FUNCTION_BLOCK PAEControlModuleBase EXTENDS PAModule IMPLEMENTS IPAControlModule
VAR_INPUT
END_VAR
VAR_OUTPUT
END_VAR
VAR	
	_FaultState : PANotifyState;
	_OperatingTime : TIME;
	_SwitchingFrequency : DINT;
	_TotalAlarms : DINT;
	_TurnOnInstant : DATE_AND_TIME;
	_TurnOffInstant : DATE_AND_TIME;
	_OnTime : TIME;
	_TurnOnDelay : TIME;
	_TurnOffDelay : TIME;
	_FaultDelayTime : TIME;
	_TurnOnInterlockDelay : TIME;
	_DepletingTime : TIME;
	_OnSiteTurnedOn : BOOL;
	_TurnOnInterlock : BOOL;
	_RunningTime : TIME;	
	_IsTriggered : BOOL;
	_FaultStateACK : BOOL;	
	_AllocatedByWay : BYTE;	
	
	// Gibt an, dass dieses Steuerungsmodul gerade von einer Funktion verwendet wird
	_AllocatedByFunction : IPAProcessFunction;
	_RoutingStateThis : PARoutingState;
	_TimerTurnOnDelay : TON;
	_TimerTurnOffDelay : TON;
END_VAR

METHOD PUBLIC AcknowledgeAlarms
VAR_INPUT
END_VAR
END_METHOD

{attribute 'TcRpcEnable'}
PROPERTY PUBLIC AllocatedByFunction : IPAProcessFunction
GET
AllocatedByFunction := _AllocatedByFunction;
END_GET
SET // PUBLIC
_AllocatedByFunction := AllocatedByFunction;
_AllocatedByWay := BOOL_TO_BYTE(_AllocatedByFunction <> 0);
Root.OnPropertyChangedByte(THIS^, 24, _AllocatedByWay);
END_SET
END_PROPERTY

{attribute 'TcRpcEnable'}
PROPERTY PUBLIC AllocatedByWay : BOOL
GET
AllocatedByWay := _AllocatedByFunction <> 0;
END_GET
END_PROPERTY

METHOD PUBLIC CombineRoutingStates : PARoutingState
VAR_INPUT
	direction : PARoutingDirection;
	rStateOfDependents : PARoutingState;
END_VAR
VAR
	rStateCombined : PARoutingState;
END_VAR
IF direction = PARoutingDirection.ToPredecessors THEN
	// TODO: Logik nochmals checken:
	IF rStateOfDependents <= PARoutingState.WaitOnPredecessors THEN
		rStateCombined := PARoutingState.WaitOnPredecessors;
	ELSE
		IF _RoutingStateThis < PARoutingState.PredecessorsFinished THEN
			rStateCombined := PARoutingState.PredecessorsFinished;
		ELSE
			rStateCombined := _RoutingStateThis;
		END_IF
	END_IF
ELSE // direction = PARoutingDirection.ToSuccessors
	IF rStateOfDependents <= PARoutingState.ReachedOnPosition THEN
		rStateCombined := PARoutingState.WaitOnSuccessor;
	ELSE //IF rStateAll >= PARoutingState.RoutePlaced THEN
		IF _RoutingStateThis = PARoutingState.ReachedOnPosition THEN
			rStateCombined := PARoutingState.RoutePlaced;
		ELSIF _RoutingStateThis <= PARoutingState.SuccessorsPlaced THEN
			rStateCombined := PARoutingState.SuccessorsPlaced;
		ELSE
			rStateCombined := _RoutingStateThis;
		END_IF
	END_IF
END_IF

CombineRoutingStates := rStateCombined;
END_METHOD

{attribute 'monitoring' := 'call'}
//{attribute 'TcRpcEnable'}
PROPERTY PUBLIC DepletingTime : TIME
GET
DepletingTime := _DepletingTime;
END_GET
SET
_DepletingTime := DepletingTime;
Root.OnPropertyChangedTime(THIS^, 22, _DepletingTime);
END_SET
END_PROPERTY

{attribute 'monitoring' := 'call'}
//{attribute 'TcRpcEnable'}
PROPERTY PUBLIC FaultDelayTime : TIME
GET
FaultDelayTime := _FaultDelayTime;
END_GET
SET
_FaultDelayTime := FaultDelayTime;
Root.OnPropertyChangedTime(THIS^, 20, _FaultDelayTime);
END_SET
END_PROPERTY

{attribute 'monitoring' := 'call'}
//{attribute 'TcRpcEnable'}
PROPERTY PUBLIC FaultState : PANotifyState
GET
FaultState := _FaultState;
END_GET
SET
_FaultState := FaultState;
Root.OnPropertyChangedInt(THIS^, 23, _FaultState);
END_SET
END_PROPERTY

{attribute 'monitoring' := 'call'}
//{attribute 'TcRpcEnable'}
PROPERTY PUBLIC FaultStateACK : BOOL
GET
FaultStateACK := _FaultStateACK;
END_GET
SET
_FaultStateACK := FaultStateACK;
Root.OnPropertyChangedBool(THIS^, 29, _FaultStateACK);
END_SET
END_PROPERTY

METHOD PUBLIC FB_postinit
VAR_INPUT
		root : IACVariobatch;
END_VAR
SUPER^.FB_postinit(root);
root.OnPropertyChangedTime(THIS^, 12, _OperatingTime);
root.OnPropertyChangedDInt(THIS^, 13, _SwitchingFrequency);
root.OnPropertyChangedDInt(THIS^, 14, _TotalAlarms);
root.OnPropertyChangedDT(THIS^, 15, _TurnOnInstant);
root.OnPropertyChangedDT(THIS^, 16, _TurnOffInstant);
root.OnPropertyChangedTime(THIS^, 17, _OnTime);
root.OnPropertyChangedTime(THIS^, 18, _TurnOnDelay);
root.OnPropertyChangedTime(THIS^, 19, _TurnOffDelay);
root.OnPropertyChangedTime(THIS^, 20, _FaultDelayTime);
root.OnPropertyChangedTime(THIS^, 21, _TurnOnInterlockDelay);
root.OnPropertyChangedTime(THIS^, 22, _DepletingTime);
root.OnPropertyChangedInt(THIS^, 23, _FaultState);
root.OnPropertyChangedByte(THIS^, 24, _AllocatedByWay);
root.OnPropertyChangedBool(THIS^, 25, _OnSiteTurnedOn);
root.OnPropertyChangedBool(THIS^, 26, _TurnOnInterlock);
root.OnPropertyChangedTime(THIS^, 27, _RunningTime);
root.OnPropertyChangedBool(THIS^, 28, _IsTriggered);
root.OnPropertyChangedBool(THIS^, 29, _FaultStateACK);
END_METHOD

// Gibt die Punkte zurück, über die die aktuelle Route gestellt ist bzw. gestellt werden soll
METHOD PUBLIC GetActivePoints : BOOL
VAR_IN_OUT
	resultPoints : ARRAY [1..GCL.cPointMAX] OF IACPoint;
END_VAR
VAR_INPUT
	pointType : PAFindPointType;
END_VAR
VAR
	i: INT;
	j: INT;
	edge : IACEdge;
	rStateAll : PARoutingState;
	iControlModule : IPAControlModule;
END_VAR
IF NOT AllocatedByWay THEN
	GetActivePoints := FALSE;
	RETURN;
END_IF

// Array leeren
FOR i:=1 TO GCL.cPointMAX BY 1
  DO
	resultPoints[i] := 0;
END_FOR;

j := 1;
// Durchlaufe alle Punkte und ermittle den Gesamtstatus über aller Nachfolgeelemente
FOR i:=1 TO GCL.cPointMAX BY 1
  DO
    IF _Points[i] <> 0 THEN
		
	    // Suche aktiven Weg
		edge := _Points[i].GetAllocatedEdge(AllocatedByFunction);
		
		IF edge <> 0 THEN
			IF (pointType = PAFindPointType.InPoints) AND (edge.Target = _Points[i]) THEN
				resultPoints[j] := _Points[i];
			ELSIF (pointType = PAFindPointType.OutPoints) AND (edge.Source = _Points[i]) THEN
				resultPoints[j] := _Points[i];
			ELSE
				resultPoints[j] := _Points[i];			
			END_IF
			j := j + 1;
		END_IF
	ELSE
		EXIT;
	END_IF
END_FOR;

GetActivePoints := TRUE;
RETURN;
END_METHOD

METHOD PUBLIC GetRoutingStateOfDependents : PARoutingState
VAR_IN_OUT
	activeOutPoints : ARRAY [1..GCL.cPointMAX] OF IACPoint;
	activeInPoints : ARRAY [1..GCL.cPointMAX] OF IACPoint;
END_VAR
VAR_INPUT
	direction : PARoutingDirection;
END_VAR
VAR
	i: INT;
	edge : IACEdge;
	rStateAll : PARoutingState;
	iControlModule : IPAControlModule;
	iProcessModule : IPAProcessModule;
	targetRoutingState : PARoutingState;
	findPointType : PAFindPointType;
END_VAR
IF NOT AllocatedByWay THEN
	GetRoutingStateOfDependents := PARoutingState.Idle;
	RETURN;
END_IF

IF direction = PARoutingDirection.ToPredecessors THEN
	findPointType := PAFindPointType.InPoints;
	rStateAll := PARoutingState.ReachedOffPosition;
ELSE // direction = PARoutingDirection.ToSuccessors
	findPointType := PAFindPointType.OutPoints;
	rStateAll := PARoutingState.RoutePlaced;
END_IF

GetActivePoints(activeOutPoints,PAFindPointType.OutPoints);
GetActivePoints(activeInPoints,PAFindPointType.InPoints);

// Durchlaufe alle Punkte und ermittle den Gesamtstatus über alle Elemente
// Falls Suchrichtung zu Nachfolger (Ausgangspunkte)
IF (direction = PARoutingDirection.ToSuccessors) THEN		
	FOR i:=1 TO GCL.cPointMAX BY 1
	  DO
		IF activeOutPoints[i] <> 0 THEN
			
			// Suche aktiven Weg
			edge := activeOutPoints[i].GetAllocatedEdge(AllocatedByFunction);
			
			// Falls das Ziel ein Control-Module ist dann frage Status ab und korrigiere Gesamtstatus aller Nachfolger
			IF __QUERYINTERFACE(edge.Target, iControlModule) THEN
				targetRoutingState := iControlModule.RoutingStateToTarget;
				IF targetRoutingState < rStateAll THEN
					rStateAll := targetRoutingState;
				END_IF
			ELSIF __QUERYINTERFACE(edge.Target, iProcessModule) THEN
				targetRoutingState := iProcessModule.RoutingStateToTarget(THIS^, rStateAll);
				IF targetRoutingState < rStateAll THEN
					rStateAll := targetRoutingState;
				END_IF
			END_IF
		ELSE
			EXIT;
		END_IF
	END_FOR;
ELSE
	FOR i:=1 TO GCL.cPointMAX BY 1
	  DO
		IF activeInPoints[i] <> 0 THEN
			
			// Suche aktiven Weg
			edge := activeInPoints[i].GetAllocatedEdge(AllocatedByFunction);
			
			// Falls das Quelle ein Control-Module ist dann frage Status ab und korrigiere Gesamtstatus aller Vorgänger
			IF __QUERYINTERFACE(edge.Source, iControlModule) THEN
				targetRoutingState := iControlModule.RoutingStateFromSource;
				IF targetRoutingState < rStateAll THEN
					rStateAll := targetRoutingState;
				END_IF
			ELSIF __QUERYINTERFACE(edge.Source, iProcessModule) THEN
				targetRoutingState := iProcessModule.RoutingStateFromSource(THIS^, rStateAll);
				IF targetRoutingState < rStateAll THEN
					rStateAll := targetRoutingState;
				END_IF
			END_IF
		ELSE
			EXIT;
		END_IF
	END_FOR;
END_IF

GetRoutingStateOfDependents := rStateAll;
END_METHOD

METHOD PUBLIC HasPointReachedOffPosition : BOOL
VAR_INPUT
	point : IACPoint;
END_VAR
HasPointReachedOffPosition := FALSE;
END_METHOD

METHOD PUBLIC HasPointReachedOnPosition : BOOL
VAR_INPUT
	point : IACPoint;
END_VAR
HasPointReachedOnPosition := FALSE;
END_METHOD

METHOD PUBLIC HavePointsReachedOffPosition : BOOL
VAR_INPUT
	activeOutPoints : ARRAY [1..GCL.cPointMAX] OF IACPoint;
	activeInPoints : ARRAY [1..GCL.cPointMAX] OF IACPoint;
END_VAR

VAR
	i: INT;
END_VAR
FOR i:=1 TO GCL.cPointMAX BY 1
  DO
    IF activeOutPoints[i] <> 0 THEN
		IF NOT HasPointReachedOffPosition(activeOutPoints[i]) THEN
			HavePointsReachedOffPosition := FALSE;
			RETURN;
		END_IF
	ELSE
		EXIT;
	END_IF
END_FOR;
FOR i:=1 TO GCL.cPointMAX BY 1
  DO
    IF activeInPoints[i] <> 0 THEN
		IF NOT HasPointReachedOffPosition(activeInPoints[i]) THEN
			HavePointsReachedOffPosition := FALSE;
			RETURN;
		END_IF
	ELSE
		EXIT;
	END_IF
END_FOR;HavePointsReachedOffPosition := TRUE;
END_METHOD

METHOD PUBLIC HavePointsReachedOnPosition : BOOL
VAR_INPUT
	activeOutPoints : ARRAY [1..GCL.cPointMAX] OF IACPoint;
	activeInPoints : ARRAY [1..GCL.cPointMAX] OF IACPoint;
END_VAR

VAR
	i: INT;
END_VAR
FOR i:=1 TO GCL.cPointMAX BY 1
  DO
    IF activeOutPoints[i] <> 0 THEN
		IF NOT HasPointReachedOnPosition(activeOutPoints[i]) THEN
			HavePointsReachedOnPosition := FALSE;
			RETURN;
		END_IF
	ELSE
		EXIT;
	END_IF
END_FOR;
FOR i:=1 TO GCL.cPointMAX BY 1
  DO
    IF activeInPoints[i] <> 0 THEN
		IF NOT HasPointReachedOnPosition(activeInPoints[i]) THEN
			HavePointsReachedOnPosition := FALSE;
			RETURN;
		END_IF
	ELSE
		EXIT;
	END_IF
END_FOR;
HavePointsReachedOnPosition := TRUE;
END_METHOD

METHOD PUBLIC InvokeSetterBool
VAR_INPUT
	PropertyID : INT;
	PropertyValue : BOOL;
END_VAR
SUPER^.InvokeSetterBool(PropertyID, PropertyValue);
CASE PropertyID OF
	25:
		OnSiteTurnedOn := PropertyValue;
	26:
		TurnOnInterlock := PropertyValue;
	28:
		IsTriggered := PropertyValue;
	29:
		FaultStateACK := PropertyValue;
END_CASE
END_METHOD

METHOD PUBLIC InvokeSetterByte
VAR_INPUT
	PropertyID : INT;
	PropertyValue : BYTE;
END_VAR
SUPER^.InvokeSetterByte(PropertyID, PropertyValue);
IF PropertyID = 24 THEN
	_AllocatedByWay := PropertyValue;
END_IF
END_METHOD

METHOD PUBLIC InvokeSetterDInt
VAR_INPUT
	PropertyID : INT;
	PropertyValue : DINT;
END_VAR
SUPER^.InvokeSetterDInt(PropertyID, PropertyValue);
CASE PropertyID OF
	13:
		SwitchingFrequency := PropertyValue;
	14:
		TotalAlarms := PropertyValue;
END_CASE
END_METHOD

METHOD PUBLIC InvokeSetterDT
VAR_INPUT
	PropertyID : INT;
	PropertyValue : DINT;
END_VAR
SUPER^.InvokeSetterDT(PropertyID, PropertyValue);
CASE PropertyID OF
	16:
		TurnOnInstant := TO_DT(PropertyValue);
	17:
		TurnOffInstant := TO_DT(PropertyValue);
END_CASE
END_METHOD

METHOD PUBLIC InvokeSetterEnum
VAR_INPUT
	PropertyID : INT;
	PropertyValue : INT;
END_VAR
SUPER^.InvokeSetterEnum(PropertyID, PropertyValue);
IF PropertyID = 23 THEN
	THIS^.FaultState := PropertyValue;
END_IF
END_METHOD

METHOD PUBLIC InvokeSetterInt
VAR_INPUT
	PropertyID : INT;
	PropertyValue : INT;
END_VAR
SUPER^.InvokeSetterInt(PropertyID, PropertyValue);
CASE PropertyID OF
	23:
		FaultState := PropertyValue;
END_CASE
END_METHOD

METHOD PUBLIC InvokeSetterTime
VAR_INPUT
	PropertyID : INT;
	PropertyValue : DINT;
END_VAR
SUPER^.InvokeSetterTime(PropertyID, PropertyValue);
CASE PropertyID OF
	12:
		OperatingTIme := TO_TIME(PropertyValue);
	17:
		OnTime := TO_TIME(PropertyValue);
	18:
		TurnOnDelay := TO_TIME(PropertyValue);
	19:
		TurnOffDelay := TO_TIME(PropertyValue);
	20:
		FaultDelayTime := TO_TIME(PropertyValue);
	21:
		TurnOnInterlockDelay := TO_TIME(PropertyValue);
	22:
		DepletingTime := TO_TIME(PropertyValue);
	27:
		RunningTime := TO_TIME(PropertyValue);
END_CASE
END_METHOD

{attribute 'monitoring' := 'call'}
//{attribute 'TcRpcEnable'}
PROPERTY PUBLIC IsTriggered : BOOL
GET
IsTriggered := _IsTriggered;
END_GET
SET
_IsTriggered := IsTriggered;
Root.OnPropertyChangedBool(THIS^,28,_IsTriggered);
END_SET
END_PROPERTY

METHOD OnInitMemory
VAR_INPUT
		root : IACVariobatch;
END_VAR
RegisterProperty(root, 12, GCL.cSizeTIME); // _OperatingTime
RegisterProperty(root, 13, GCL.cSizeDINT); // _SwitchingFrequency
RegisterProperty(root, 14, GCL.cSizeDINT); // _TotalAlarms
RegisterProperty(root, 15, GCL.cSizeDT); // _TurnOnInstant
RegisterProperty(root, 16, GCL.cSizeDT); // _TurnOffInstant
RegisterProperty(root, 17, GCL.cSizeTIME); // _OnTime
RegisterProperty(root, 18, GCL.cSizeTIME); // TurnOnDelay
RegisterProperty(root, 19, GCL.cSizeTIME); // TurnOffDelay
RegisterProperty(root, 20, GCL.cSizeTIME); // FaultDelayTime
RegisterProperty(root, 21, GCL.cSizeTIME); // TurnOnInterlockDelay
RegisterProperty(root, 22, GCL.cSizeTIME); // DepletingTime
RegisterProperty(root, 23, GCL.cSizeINT); // FaultState
RegisterProperty(root, 24, GCL.cSizeBYTE); // AllocatedByWay
RegisterProperty(root, 25, GCL.cSizeBYTE); // OnSiteTurnedOn
RegisterProperty(root, 26, GCL.cSizeBYTE); // TurnOnInterlock
RegisterProperty(root, 27, GCL.cSizeTIME); // RunningTime
RegisterProperty(root, 28, GCL.cSizeBYTE); // IsTriggered
RegisterProperty(root, 29, GCL.cSizeBYTE); // FaultStateACK
SUPER^.OnInitMemory(root);
END_METHOD

METHOD PROTECTED OnMainEnter
VAR_INPUT
END_VAR
VAR
	activePoints : ARRAY [1..GCL.cPointMAX] OF IACPoint;
	rStateOfDependents : PARoutingState;
END_VAR
SUPER^.OnMainEnter();
IF AllocatedByWay THEN
	CASE AllocatedByFunction.ACState OF
		//ACStateEnum.SMIdle:
		//ACStateEnum.SMStarting:

		ACStateEnum.SMRunning:
			SMStartAndControlWithDelay();
		
		//ACStateEnum.SMCompleted:
		//ACStateEnum.SMResetting:
		
		ACStateEnum.SMPausing:
			SMStopIntermediately();
		//ACStateEnum.SMPaused:
		ACStateEnum.SMResuming:
			SMStartAndControlIntermediately();
		
		ACStateEnum.SMHolding:
			SMStopWithDelay();
		//ACStateEnum.SMHeld:	
		ACStateEnum.SMRestarting:
			SMStartAndControlWithDelay();
			
		ACStateEnum.SMAborting:
			SMStopIntermediately();
		//ACStateEnum.SMAborted:
		
		ACStateEnum.SMStopping:
			SMStopWithDelay();
		//ACStateEnum.SMStopped:
	END_CASE
END_IF
END_METHOD

{attribute 'monitoring' := 'call'}
//{attribute 'TcRpcEnable'}
PROPERTY PUBLIC OnSiteTurnedOn : BOOL
GET
OnSiteTurnedOn := _OnSiteTurnedOn;
END_GET
SET
_OnSiteTurnedOn := OnSiteTurnedOn;
Root.OnPropertyChangedBool(THIS^, 25, _OnSiteTurnedOn);
END_SET
END_PROPERTY

{attribute 'monitoring' := 'call'}
//{attribute 'TcRpcEnable'}
PROPERTY PUBLIC OnTime : TIME
GET
OnTime := _OnTime;
END_GET
SET
_OnTime := OnTime;
Root.OnPropertyChangedTime(THIS^, 17, _OnTime);
END_SET
END_PROPERTY

{attribute 'monitoring' := 'call'}
//{attribute 'TcRpcEnable'}
PROPERTY OperatingTime : TIME
GET
OperatingTime := _OperatingTime;
END_GET
SET
_OperatingTime := OperatingTime;
Root.OnPropertyChangedTime(THIS^, 12, _OperatingTime);
END_SET
END_PROPERTY

PROPERTY RoutingStateFromSource : PARoutingState
GET
VAR
	rStateOfDependents : PARoutingState;
	rStateCombined : PARoutingState;
END_VAR
IF NOT AllocatedByWay THEN
	RoutingStateFromSource := PARoutingState.Idle;
	RETURN;
END_IF

rStateOfDependents := RoutingStateOfPredecessors;
rStateCombined := CombineRoutingStates(PARoutingDirection.ToPredecessors, rStateOfDependents);
RoutingStateFromSource := rStateCombined;
END_GET
END_PROPERTY

PROPERTY RoutingStateOfPredecessors : PARoutingState
GET
VAR
	activeOutPoints : ARRAY [1..GCL.cPointMAX] OF IACPoint;
	activeInPoints : ARRAY [1..GCL.cPointMAX] OF IACPoint;
	rStateAll : PARoutingState;
END_VAR
IF NOT AllocatedByWay THEN
	RoutingStateOfPredecessors := PARoutingState.Idle;
	RETURN;
END_IF

rStateAll := GetRoutingStateOfDependents(activeOutPoints,activeInPoints,PARoutingDirection.ToPredecessors);
RoutingStateOfPredecessors := rStateAll;
END_GET
END_PROPERTY

PROPERTY RoutingStateOfSuccessors : PARoutingState
GET
VAR
	activeOutPoints : ARRAY [1..GCL.cPointMAX] OF IACPoint;
	activeInPoints : ARRAY [1..GCL.cPointMAX] OF IACPoint;
	rStateAll : PARoutingState;
END_VAR
IF NOT AllocatedByWay THEN
	RoutingStateOfSuccessors := PARoutingState.Idle;
	RETURN;
END_IF

rStateAll := GetRoutingStateOfDependents(activeOutPoints,activeInPoints,PARoutingDirection.ToSuccessors);
RoutingStateOfSuccessors := rStateAll;
END_GET
END_PROPERTY

PROPERTY PUBLIC RoutingStateThis : PARoutingState
GET
RoutingStateThis := _RoutingStateThis;
END_GET
END_PROPERTY

PROPERTY RoutingStateToTarget : PARoutingState
GET
VAR
	rStateOfDependents : PARoutingState;
	rStateCombined : PARoutingState;
END_VAR
IF NOT AllocatedByWay THEN
	RoutingStateToTarget := PARoutingState.Idle;
	RETURN;
END_IF

rStateOfDependents := RoutingStateOfSuccessors;
rStateCombined := CombineRoutingStates(PARoutingDirection.ToSuccessors, rStateOfDependents);
RoutingStateToTarget := rStateCombined;
END_GET
END_PROPERTY

{attribute 'monitoring' := 'call'}
//{attribute 'TcRpcEnable'}
PROPERTY PUBLIC RunningTime : TIME
GET
RunningTime := _RunningTime;
END_GET
SET
_RunningTime := RunningTime;
Root.OnPropertyChangedTime(THIS^, 27, _RunningTime);
END_SET
END_PROPERTY

// Weg anfahren ohne Zeiten und anschliessend Weg überwachen. (Falls Nachfolgelemente angehalten, dann auch selbst anhalten)
METHOD PROTECTED SMStartAndControlIntermediately
VAR
	activeOutPoints : ARRAY [1..GCL.cPointMAX] OF IACPoint;
	activeInPoints : ARRAY [1..GCL.cPointMAX] OF IACPoint;
	rStateOfDependents : PARoutingState;
END_VAR
rStateOfDependents := THIS^.GetRoutingStateOfDependents(activeOutPoints, activeInPoints, PARoutingDirection.ToSuccessors);
IF (rStateOfDependents = PARoutingState.RoutePlaced) THEN
	
	IF (THIS^._RoutingStateThis <= PARoutingState.TurnOnElapsing) OR (THIS^._RoutingStateThis >= PARoutingState.WaitOnPredecessors) THEN
		THIS^._RoutingStateThis := PARoutingState.MovingOrTurningOn;
	END_IF
	
	IF THIS^._RoutingStateThis = PARoutingState.MovingOrTurningOn THEN
		IF HavePointsReachedOnPosition(activeOutPoints, activeInPoints) THEN
			THIS^._RoutingStateThis := PARoutingState.ReachedOnPosition;
		END_IF
		RETURN;
	END_IF
ELSE
	_TimerTurnOnDelay.IN := FALSE;
	THIS^._RoutingStateThis := PARoutingState.WaitOnSuccessor;
END_IF
END_METHOD

// Weg anfahren mit Zeiten und anschliessend Weg überwachen. (Falls Nachfolgelemente angehalten, dann auch selbst anhalten)
METHOD PROTECTED SMStartAndControlWithDelay
VAR
	activeOutPoints : ARRAY [1..GCL.cPointMAX] OF IACPoint;
	activeInPoints : ARRAY [1..GCL.cPointMAX] OF IACPoint;
	rStateOfDependents : PARoutingState;
END_VAR
rStateOfDependents := THIS^.GetRoutingStateOfDependents(activeOutPoints, activeInPoints, PARoutingDirection.ToSuccessors);
IF (rStateOfDependents = PARoutingState.RoutePlaced) THEN
	
	IF (THIS^._RoutingStateThis < PARoutingState.TurnOnElapsing) OR (THIS^._RoutingStateThis >= PARoutingState.WaitOnPredecessors) THEN
		_TimerTurnOnDelay(IN := TRUE,PT := TurnOnDelay);
		THIS^._RoutingStateThis := PARoutingState.TurnOnElapsing;
	END_IF	
	
	IF THIS^._RoutingStateThis = PARoutingState.TurnOnElapsing THEN
		IF (_TimerTurnOnDelay.Q) THEN
			THIS^._RoutingStateThis := PARoutingState.MovingOrTurningOn;
		ELSE
			RETURN;
		END_IF
	END_IF
	
	IF THIS^._RoutingStateThis = PARoutingState.MovingOrTurningOn THEN
		IF HavePointsReachedOnPosition(activeOutPoints, activeInPoints) THEN
			THIS^._RoutingStateThis := PARoutingState.ReachedOnPosition;
		END_IF
	END_IF
ELSE
	_TimerTurnOnDelay.IN := FALSE;
	THIS^._RoutingStateThis := PARoutingState.WaitOnSuccessor;
END_IF
END_METHOD

// Weg unverzüglich anhalten
METHOD PROTECTED SMStopIntermediately
VAR
	activeOutPoints : ARRAY [1..GCL.cPointMAX] OF IACPoint;
	activeInPoints : ARRAY [1..GCL.cPointMAX] OF IACPoint;
	rStateOfDependents : PARoutingState;
END_VAR
rStateOfDependents := THIS^.GetRoutingStateOfDependents(activeOutPoints, activeInPoints, PARoutingDirection.ToPredecessors);
IF (rStateOfDependents = PARoutingState.ReachedOffPosition) THEN
	
	IF THIS^._RoutingStateThis <= PARoutingState.TurnOffElapsing THEN
		THIS^._RoutingStateThis := PARoutingState.MovingOrTurningOff;
	END_IF	
	
	IF THIS^._RoutingStateThis = PARoutingState.MovingOrTurningOff THEN
		IF HavePointsReachedOffPosition(activeOutPoints, activeInPoints) THEN
			THIS^._RoutingStateThis := PARoutingState.ReachedOffPosition;
		END_IF
	END_IF
ELSE
	_TimerTurnOffDelay.IN := FALSE;
	THIS^._RoutingStateThis := PARoutingState.WaitOnPredecessors;
END_IF
END_METHOD

// Weg abfahren mit Zeiten.
METHOD PROTECTED SMStopWithDelay
VAR
	activeOutPoints : ARRAY [1..GCL.cPointMAX] OF IACPoint;
	activeInPoints : ARRAY [1..GCL.cPointMAX] OF IACPoint;
	rStateOfDependents : PARoutingState;
END_VAR
rStateOfDependents := THIS^.GetRoutingStateOfDependents(activeOutPoints, activeInPoints, PARoutingDirection.ToPredecessors);
IF (rStateOfDependents = PARoutingState.ReachedOffPosition) THEN
	
	IF THIS^._RoutingStateThis < PARoutingState.TurnOffElapsing THEN
		_TimerTurnOffDelay(IN := TRUE,PT := TurnOffDelay);
		THIS^._RoutingStateThis := PARoutingState.TurnOffElapsing;
	END_IF	
	
	IF THIS^._RoutingStateThis = PARoutingState.TurnOffElapsing THEN
		IF (_TimerTurnOffDelay.Q) THEN
			THIS^._RoutingStateThis := PARoutingState.MovingOrTurningOff;
		ELSE
			RETURN;
		END_IF
	END_IF
	
	IF THIS^._RoutingStateThis = PARoutingState.MovingOrTurningOff THEN
		IF HavePointsReachedOffPosition(activeOutPoints, activeInPoints) THEN
			THIS^._RoutingStateThis := PARoutingState.ReachedOffPosition;
		END_IF
	END_IF
ELSE
	_TimerTurnOffDelay.IN := FALSE;
	THIS^._RoutingStateThis := PARoutingState.WaitOnPredecessors;
END_IF
END_METHOD

{attribute 'monitoring' := 'call'}
//{attribute 'TcRpcEnable'}
PROPERTY PUBLIC SwitchingFrequency : DINT
GET
SwitchingFrequency := _SwitchingFrequency;
END_GET
SET
_SwitchingFrequency := SwitchingFrequency;
Root.OnPropertyChangedDInt(THIS^, 13, _SwitchingFrequency);
END_SET
END_PROPERTY

{attribute 'monitoring' := 'call'}
//{attribute 'TcRpcEnable'}
PROPERTY PUBLIC TotalAlarms : DINT
GET
TotalAlarms := _TotalAlarms;
END_GET
SET
_TotalAlarms := TotalAlarms;
Root.OnPropertyChangedDInt(THIS^, 14, _TotalAlarms);
END_SET
END_PROPERTY

{attribute 'monitoring' := 'call'}
//{attribute 'TcRpcEnable'}
PROPERTY PUBLIC TurnOffDelay : TIME
GET
TurnOffDelay := _TurnOffDelay;
END_GET
SET
_TurnOffDelay := TurnOffDelay;
Root.OnPropertyChangedTime(THIS^, 19, _TurnOffDelay);
END_SET
END_PROPERTY

{attribute 'monitoring' := 'call'}
//{attribute 'TcRpcEnable'}
PROPERTY PUBLIC TurnOffInstant : DATE_AND_TIME
GET
TurnOffInstant := _TurnOffInstant;
END_GET
SET
_TurnOffInstant := TurnOffInstant;
Root.OnPropertyChangedDT(THIS^, 16, _TurnOffInstant);
END_SET
END_PROPERTY

{attribute 'monitoring' := 'call'}
//{attribute 'TcRpcEnable'}
PROPERTY PUBLIC TurnOnDelay : TIME
GET
TurnOnDelay := _TurnOnDelay;
END_GET
SET
_TurnOnDelay := TurnOnDelay;
Root.OnPropertyChangedTime(THIS^, 18, _TurnOnDelay);
END_SET
END_PROPERTY

{attribute 'monitoring' := 'call'}
//{attribute 'TcRpcEnable'}
PROPERTY PUBLIC TurnOnInstant : DATE_AND_TIME
GET
TurnOnInstant := _TurnOnInstant;
END_GET
SET
_TurnOnInstant := TurnOnInstant;
Root.OnPropertyChangedDT(THIS^, 15, _TurnOnInstant);
END_SET
END_PROPERTY

{attribute 'monitoring' := 'call'}
//{attribute 'TcRpcEnable'}
PROPERTY PUBLIC TurnOnInterlock : BOOL
GET
TurnOnInterlock := _TurnOnInterlock;
END_GET
SET
_TurnOnInterlock := TurnOnInterlock;
Root.OnPropertyChangedBool(THIS^, 26, _TurnOnInterlock);
END_SET
END_PROPERTY

{attribute 'monitoring' := 'call'}
//{attribute 'TcRpcEnable'}
PROPERTY PUBLIC TurnOnInterlockDelay : TIME
GET
TurnOnInterlockDelay := _TurnOnInterlockDelay;
END_GET
SET
_TurnOnInterlockDelay := TurnOnInterlockDelay;
Root.OnPropertyChangedTime(THIS^, 21, _TurnOnInterlockDelay);
END_SET
END_PROPERTY

END_FUNCTION_BLOCK

(* stored: Version 1.1.0.1, ProductVersion 3.1.4024.6
   POU PAEControlModuleBase: Id {a756d94a-22c1-470e-b3c0-dd546f11be3d}, SpecialFunc None
   Folder ModuleProperties: Id {f78ca878-981c-4622-a41e-101a9f8e7f2f}
   Folder Routing: Id {a5ecdbcf-3d11-41ee-8ab9-6f65c0eff01a}
   Folder StateHandling: Id {863f9ed5-4617-4c9f-a590-db3f72f2cbc1}
   Method AcknowledgeAlarms: Id {762dcf9d-49cc-42f9-90a0-cc524c1678e6}
   Property AllocatedByFunction: Id {762b0cb6-cc24-4bd5-ae84-85a8f48ae51b}
   Get Get: Id {7d82c250-20cf-4a66-977f-6fc43a25d44d}
   Set Set: Id {940013ec-c7c5-4523-a327-1c056ba5f865}
   Property AllocatedByWay: Id {9ba54cea-c52b-4502-b703-28fed5f5f7f8}
   Get Get: Id {33ac9d79-c140-44d7-ad61-72f12cdff5e4}
   Method CombineRoutingStates: Id {8cbd8a75-66f4-4b22-a9d4-8b8ac1b359b9}
   Property DepletingTime: Id {0d6193f0-77f2-4a7c-a4dd-9768daec3608}
   Get Get: Id {b8c03518-5d89-4c88-a6c1-a2b72560aad6}
   Set Set: Id {b4217e4b-3cac-4aaf-b0b8-c3b5af428b33}
   Property FaultDelayTime: Id {585ce37b-8d38-4e4e-81f7-8519b6d9f7ee}
   Get Get: Id {7237680e-374f-45da-955a-41cb7695bfa8}
   Set Set: Id {0802c52c-2875-453c-b2f8-70fca73792b8}
   Property FaultState: Id {e9212465-70f5-42b0-8bee-f8d788d43ba9}
   Get Get: Id {989edf0f-f4a1-4990-a75e-5a4e51e3bbf2}
   Set Set: Id {208b89c9-78c8-4db2-b157-41f4573c5f7a}
   Property FaultStateACK: Id {61499a33-6823-4cb9-ba73-0268de49e6f7}
   Get Get: Id {c5760855-b065-40cf-8b78-b108b2ae004f}
   Set Set: Id {74a40647-fbe4-43b7-b759-08aa85eef81e}
   Method FB_postinit: Id {8e469907-4f38-4d99-96b3-cc6d1dd85cb7}
   Method GetActivePoints: Id {8255df67-529b-4e6f-a19c-c146969fb1fa}
   Method GetRoutingStateOfDependents: Id {f9893d72-3c41-45cf-be8b-b606d2a7c51f}
   Method HasPointReachedOffPosition: Id {d5381425-48dc-44b3-b482-92c59ac6da5c}
   Method HasPointReachedOnPosition: Id {15c6ef5a-8bf7-4951-901d-7956b337ece7}
   Method HavePointsReachedOffPosition: Id {6cd5ea6a-b101-4d97-9a5d-35f2634c0640}
   Method HavePointsReachedOnPosition: Id {2f5b89de-6523-4cc2-bcb1-f54654d95130}
   Method InvokeSetterBool: Id {363794f5-ce67-4811-8a82-c4bffa2ea76c}
   Method InvokeSetterByte: Id {cb0b5ea7-9ca4-42d3-9609-61bcdb644464}
   Method InvokeSetterDInt: Id {370b925d-5c8b-400b-b34c-e0b3147c293a}
   Method InvokeSetterDT: Id {c087178b-da4c-418e-983d-7b8d2fe6d57a}
   Method InvokeSetterEnum: Id {48c254a8-7d2a-4a2b-80ec-3031912aa597}
   Method InvokeSetterInt: Id {8be91f0d-8fe8-4ae6-947b-3b1e9c16a84a}
   Method InvokeSetterTime: Id {91b56297-798a-45e9-94cd-f8bdaefc46a0}
   Property IsTriggered: Id {7a7212b3-addc-4e77-b9cb-fe5425db76dc}
   Get Get: Id {7cb7c090-c4ff-4e53-8e2c-d5829597b5a8}
   Set Set: Id {e6b93db9-63ea-491b-82da-d267fdefd16b}
   Method OnInitMemory: Id {803ca1bf-a80b-40b9-8a20-2180636babdb}
   Method OnMainEnter: Id {23688101-43c5-475f-b683-184315c4b08d}
   Property OnSiteTurnedOn: Id {4f11b984-3c12-4fe7-963a-c86f43f22dc7}
   Get Get: Id {6afc68c9-5ceb-414b-842c-209914ed0385}
   Set Set: Id {b18a314d-ded7-49b4-af23-24065b040ce6}
   Property OnTime: Id {90931188-660d-4202-aa15-ec9cdb396638}
   Get Get: Id {c7f86e69-b119-4225-9234-57b75458d342}
   Set Set: Id {c45957b9-56b2-4761-b538-c71a4577a2ce}
   Property OperatingTime: Id {19e08576-e8f7-4555-9a73-c149f83be78d}
   Get Get: Id {e9997d58-adbb-4bb9-a749-c311f18cfcd2}
   Set Set: Id {9f2463bd-01a3-4e6a-9cb1-704f00400103}
   Property RoutingStateFromSource: Id {811632c2-1030-498a-8665-aaea9bb41082}
   Get Get: Id {c0918eab-e3cc-4458-bf32-dd0bbc259262}
   Property RoutingStateOfPredecessors: Id {cc34207b-2cff-4043-bed9-a1eb58661155}
   Get Get: Id {07cf3e47-c2ef-4f72-a004-2eccc2def3c8}
   Property RoutingStateOfSuccessors: Id {17ce9339-d5d0-4cc2-b320-018447f974d1}
   Get Get: Id {2dedf017-1666-4deb-b654-4b90f5fd6b46}
   Property RoutingStateThis: Id {bd8ee09a-2695-49d6-8ea1-604c80659027}
   Get Get: Id {82efcb33-1c8a-4566-bd23-7afa0a82c900}
   Property RoutingStateToTarget: Id {065d25f7-370b-45ac-8c23-9343c77b435b}
   Get Get: Id {3a34eb73-0159-4154-8cba-60091d97c8a7}
   Property RunningTime: Id {d7bed24e-bb15-49cd-a5a1-8bdeabffb439}
   Get Get: Id {1366aebb-bc11-45bb-99b5-5da2ffa439d4}
   Set Set: Id {34b2cea2-58a3-4bd0-8955-06afbb8d8318}
   Method SMStartAndControlIntermediately: Id {162f7d6d-8acf-48a2-8fa4-85f455f34309}
   Method SMStartAndControlWithDelay: Id {36a5888c-af1e-4efa-9280-8098093e2e23}
   Method SMStopIntermediately: Id {940ffc15-d570-43bc-b85d-8fcff5ed77c3}
   Method SMStopWithDelay: Id {41d4f2fb-b4ab-4f5f-8554-4f12c8b8c7cc}
   Property SwitchingFrequency: Id {49c106ba-27c3-4456-a6f2-a5243c35d692}
   Get Get: Id {674ccd86-0883-486e-b48e-763c60d65c36}
   Set Set: Id {ccbd352d-918c-4ca0-8496-ad3837e43632}
   Property TotalAlarms: Id {bd1aef9e-1489-442d-b0f7-dc1a1793f687}
   Get Get: Id {ec021631-ab63-4ba6-8646-2e75c79fd23e}
   Set Set: Id {ec8e4be6-77e2-4005-9bf9-0edb75344d52}
   Property TurnOffDelay: Id {8a1c3291-d173-46dc-89a6-6d7836dfedd9}
   Get Get: Id {77b89797-0748-4861-ae3f-2905e328e02f}
   Set Set: Id {47d13aac-ab6c-40ba-8c8e-ac028b72c852}
   Property TurnOffInstant: Id {b9122ac9-47a7-495c-9a01-5f4e0561ff3c}
   Get Get: Id {f5f66ec8-cb70-4f7a-a7de-6b02a0e82ca1}
   Set Set: Id {26a04a74-ce0d-4d68-b3a7-d0b1c88da6b4}
   Property TurnOnDelay: Id {a6bf0cee-2387-4fe7-b7f6-f91d3753aa0e}
   Get Get: Id {9190e59f-2f75-46ec-a25d-83a849cc1a44}
   Set Set: Id {01a7e247-1f05-4b87-85ec-a9a3dfd059d9}
   Property TurnOnInstant: Id {81ff9cf3-d020-4f30-aaa6-0cc54d4069bd}
   Get Get: Id {00dc6f98-8132-4fdb-b5e7-f6d7a1c6d5fb}
   Set Set: Id {6dce0667-c9a6-422e-9c8f-f6eacc8788d4}
   Property TurnOnInterlock: Id {ac22fc36-3519-4911-9b76-b06f76906e94}
   Get Get: Id {9c0e115c-eaa2-4a69-b072-b0e4f4b057c5}
   Set Set: Id {95a3e0b7-9683-4b53-83b9-00af0ec655c7}
   Property TurnOnInterlockDelay: Id {eb2cc891-b925-4669-80a5-7dac4c580034}
   Get Get: Id {fe1e0139-05d3-469b-bb8b-8574136fe0e3}
   Set Set: Id {243cf18d-7235-4173-840b-f0344bc6e321} *)
